Universal Robots PolyScope program: bearing_move_to_asm_hole.urp

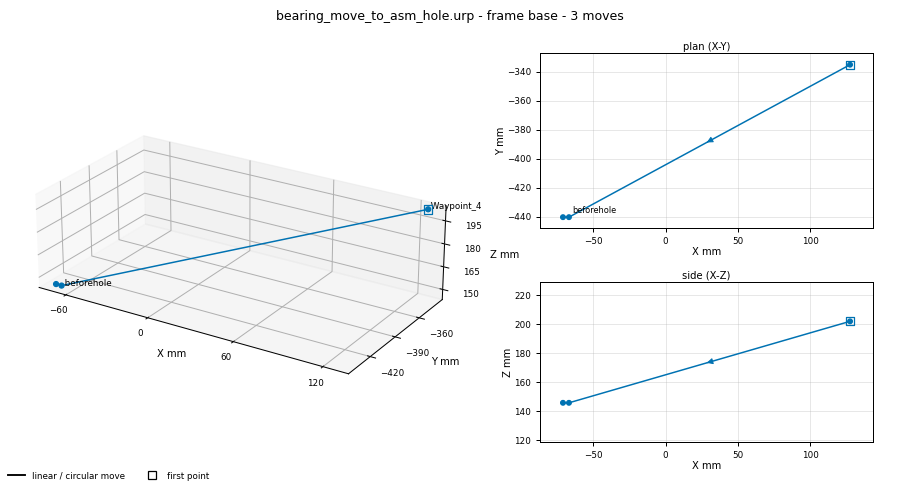
[picture p0: tool path of bearing_move_to_asm_hole.urp in frame base, 3 of 4 moves have a stored position in this frame; points joined in program order, loops and branches not executed]
Program bearing_move_to_asm_hole (installation=default directory=/programs/wrs2020 createdIn=5.7.0.90932 lastSavedIn=5.10.0.106288 robotSerialNumber=20205500607)
Calibrated DH parameters: a=[0.000096, -0.337, -0.383372, 0.000118, 0.000015, 0]; d=[0.162724, 79.377998, -95.545185, 16.300583, 0.099689, 0.099499]; alpha=[1.569249, 0.003272, 0.005201, 1.570041, -1.570219, 0]; deltaTheta=[0, 0.65664, 5.410619, 0.215927, -0.000001, 0]
Robot Program (runOnlyOnce=true)
  MoveJ speed 60 deg/s, acceleration 80 deg/s^2 (useActiveTCP=true) feature=Base
    currentpose := get_actual_joint_positions()
    Waypoint Waypoint (Variable): variable(name=currentpose)
  SuppressedNode
    MoveL speed 600 mm/s, acceleration 1200 mm/s^2 (useActiveTCP=false) tcp=gripper_85_tip; feature=Base
      Waypoint above: TCP in base x=200.55 y=-207.27 z=86.012 mm, rx=0.028 ry=3.1154 rz=0.0066 rad; joints [105.259, -116.491, 145.894, -119.54, -88.262, 16.238] deg; TCP offset x=0 y=0 z=165 mm, rx=0 ry=0 rz=0 rad
  'go to hole'
  MoveL speed 250 mm/s, acceleration 1200 mm/s^2 (useActiveTCP=false) tcp=gripper_85_tip; feature=Base
    Waypoint Waypoint_4: motionParameters(blendRadius=0.03); TCP in base x=127.347 y=-335.091 z=202.15 mm, rx=1.8898 ry=-2.0717 rz=-0.3374 rad; joints [105.843, -103.2, 121.421, -103.978, -112.085, -68.171] deg
    Waypoint beforehole: TCP in base x=-66.726 y=-440.354 z=145.893 mm, rx=1.497 ry=-1.6176 rz=-0.8285 rad; joints [94.029, -78.493, 127.683, -136.29, -150.015, -79.747] deg
    Waypoint athole: TCP in base x=-70.859 y=-440.353 z=145.897 mm, rx=1.497 ry=-1.6176 rz=-0.8285 rad; joints [93.491, -78.459, 128.002, -137.579, -150.038, -80.825] deg
